SUBAPPLICATION SoftKey_Verteiler_senken (* Subapplication Type *)
  (* Standard: 61499-2 *)
  (* Version 1.0, 2023-02-11, franz *)
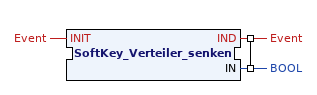
  EVENT_INPUT
    INIT;
  END_EVENT
  EVENT_OUTPUT
    IND WITH IN;
  END_EVENT
  VAR_OUTPUT
    IN : BOOL;
  END_VAR
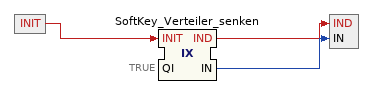
  FBS
    SoftKey_Verteiler_senken : IX(QI := TRUE);
  END_FBS
  EVENT_CONNECTIONS
    INIT TO SoftKey_Verteiler_senken.INIT;
    SoftKey_Verteiler_senken.IND TO IND;
  END_CONNECTIONS
  DATA_CONNECTIONS
    SoftKey_Verteiler_senken.IN TO IN;
  END_CONNECTIONS
END_SUBAPPLICATION
